(* Logix 5000 project; controller default_profile 5069-L306ERM rev 31.11; software revision 31.01 *)

TASK MainTask (continuous, watchdog 500 ms) : MainProgram

MODULES
   Local : 5069-L306ERM (5069 0, rev 31.11)
       : 5069-IB16 (5069 2, rev 2.14, StandardDataDriven RPI 5 ms)
       : vendor 1 type 7 code 1213 (5069 1, rev 3.14, StandardDataDriven RPI 5 ms)
END_MODULES

VAR_GLOBAL   (* controller tags *)
   Heater_Blower : BOOL;
   Load_Cell : DINT;
   Motor1_Backwards : BOOL;
   Motor1_Forwards : BOOL;
   Motor2 : BOOL;
   Motor_Timer : TIMER := (PRE := 2000);
   Piston : BOOL;
   Piston_Timer : TIMER := (PRE := 10);
   Platform_1 : DINT;
   Platform_2 : DINT := 1000000;
   Platform_3 : DINT := 2000000;
   Position : DINT;
   Radians : DINT;
   Rotation : DINT;
   RUN : BOOL;
   STANDBY : BOOL := 1;
   START : BOOL;
   STOP : BOOL;
   SV1 : BOOL;
   SV2 : BOOL;
   Task : DINT;
   Timer1 : TIMER := (PRE := 6000);
   Timer2 : TIMER := (PRE := 25000);
END_VAR

PROGRAM MainProgram   (* main routine MainRoutine *)

ROUTINE MainRoutine   (* ladder *)
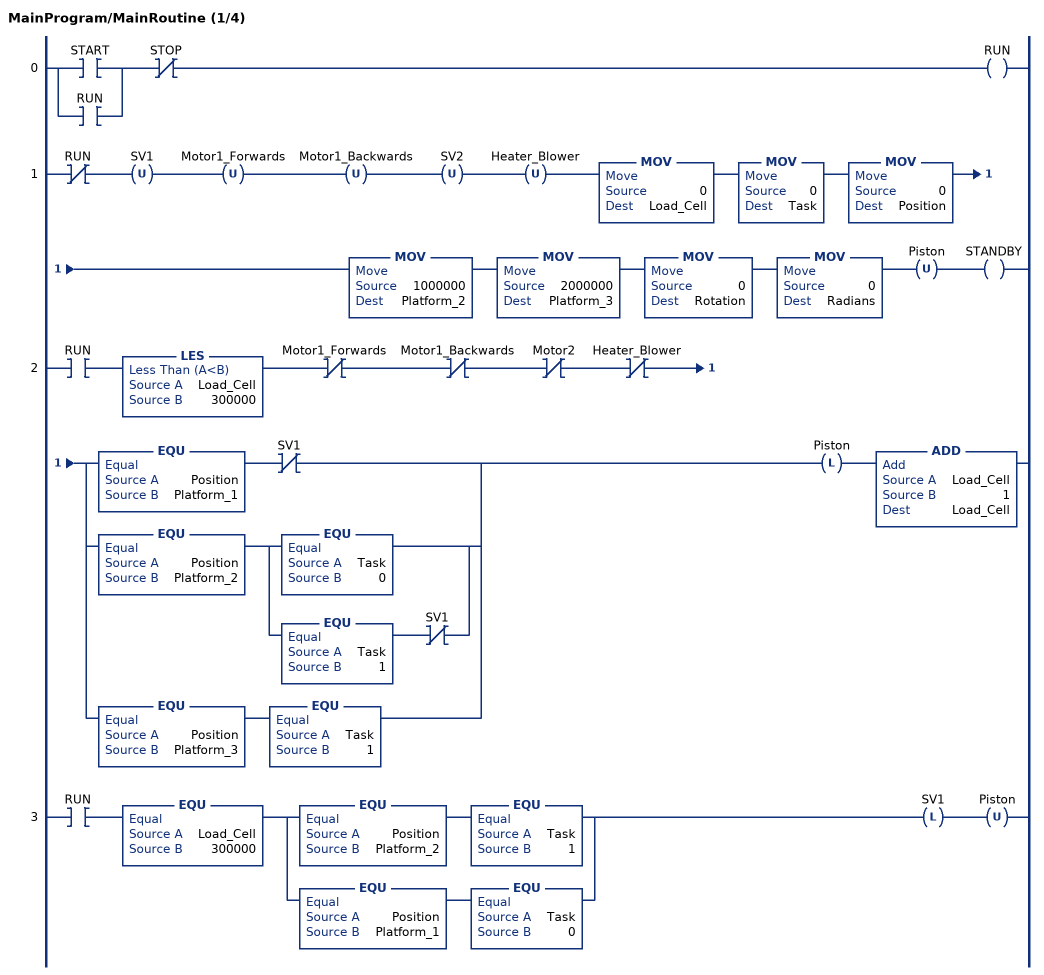
   0: [XIC(START) ,XIC(RUN) ]XIO(STOP)OTE(RUN);
   1: XIO(RUN)OTU(SV1)OTU(Motor1_Forwards)OTU(Motor1_Backwards)OTU(SV2)OTU(Heater_Blower)MOV(0,Load_Cell)MOV(0,Task)MOV(0,Position)MOV(1000000,Platform_2)MOV(2000000,Platform_3)MOV(0,Rotation)MOV(0,Radians)OTU(Piston)OTE(STANDBY);
   2: XIC(RUN)LES(Load_Cell,300000)XIO(Motor1_Forwards)XIO(Motor1_Backwards)XIO(Motor2)XIO(Heater_Blower)[EQU(Position,Platform_1) XIO(SV1) ,[EQU(Position,Platform_2) [EQU(Task,0) ,EQU(Task,1) XIO(SV1) ] ,EQU(Position,Platform_3) EQU(Task,1) ] ]OTL(Piston)ADD(Load_Cell,1,Load_Cell);
   3: XIC(RUN)EQU(Load_Cell,300000)[EQU(Position,Platform_2) EQU(Task,1) ,EQU(Position,Platform_1) EQU(Task,0) ]OTL(SV1)OTU(Piston);
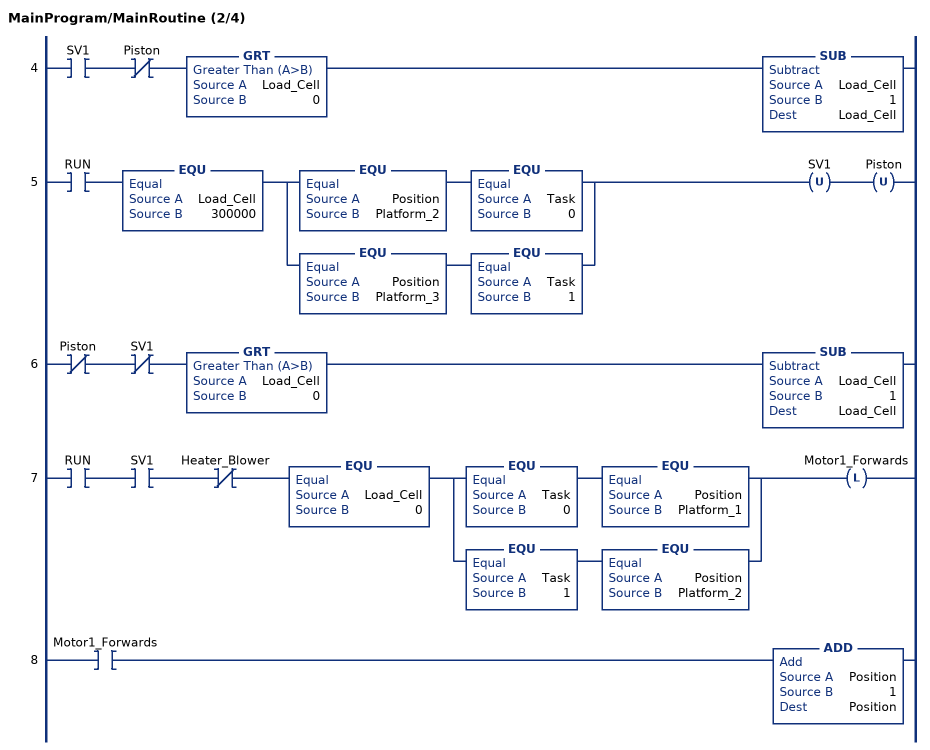
   4: XIC(SV1)XIO(Piston)GRT(Load_Cell,0)SUB(Load_Cell,1,Load_Cell);
   5: XIC(RUN)EQU(Load_Cell,300000)[EQU(Position,Platform_2) EQU(Task,0) ,EQU(Position,Platform_3) EQU(Task,1) ]OTU(SV1)OTU(Piston);
   6: XIO(Piston)XIO(SV1)GRT(Load_Cell,0)SUB(Load_Cell,1,Load_Cell);
   7: XIC(RUN)XIC(SV1)XIO(Heater_Blower)EQU(Load_Cell,0)[EQU(Task,0) EQU(Position,Platform_1) ,EQU(Task,1) EQU(Position,Platform_2) ]OTL(Motor1_Forwards);
   8: XIC(Motor1_Forwards)ADD(Position,1,Position);
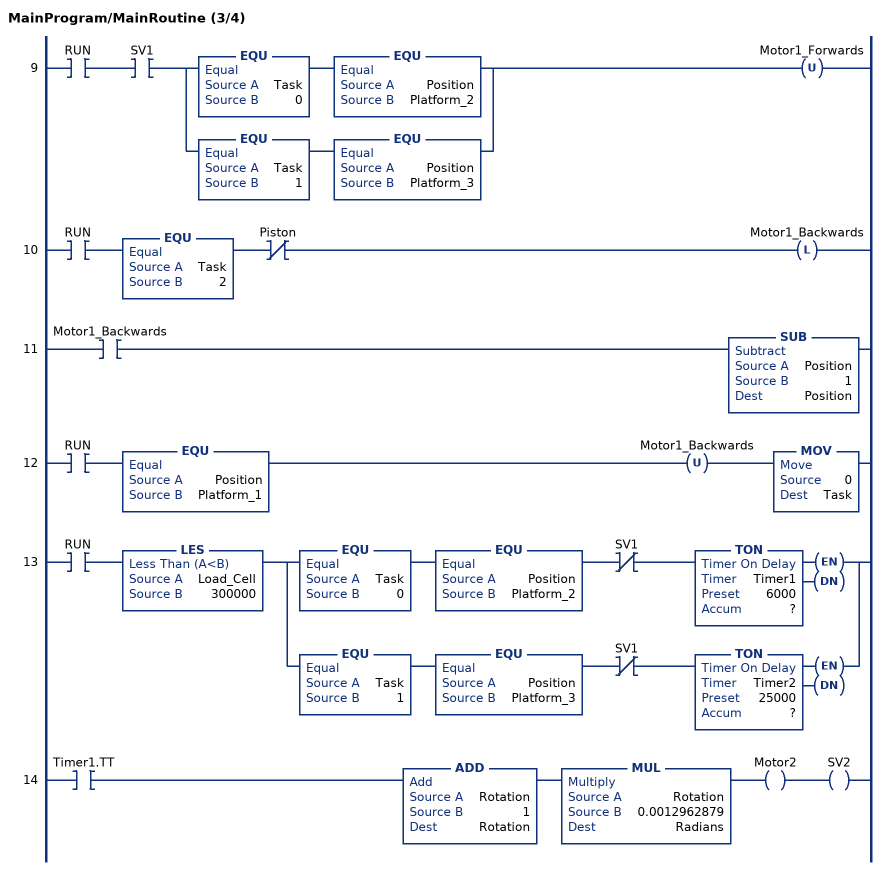
   9: XIC(RUN)XIC(SV1)[EQU(Task,0) EQU(Position,Platform_2) ,EQU(Task,1) EQU(Position,Platform_3) ]OTU(Motor1_Forwards);
   10: XIC(RUN)EQU(Task,2)XIO(Piston)OTL(Motor1_Backwards);
   11: XIC(Motor1_Backwards)SUB(Position,1,Position);
   12: XIC(RUN)EQU(Position,Platform_1)OTU(Motor1_Backwards)MOV(0,Task);
   13: XIC(RUN)LES(Load_Cell,300000)[EQU(Task,0) EQU(Position,Platform_2) XIO(SV1) TON(Timer1,?,?) ,EQU(Task,1) EQU(Position,Platform_3) XIO(SV1) TON(Timer2,?,?) ];
   14: XIC(Timer1.TT)ADD(Rotation,1,Rotation)MUL(Rotation,0.0012962879,Radians)OTE(Motor2)OTE(SV2);
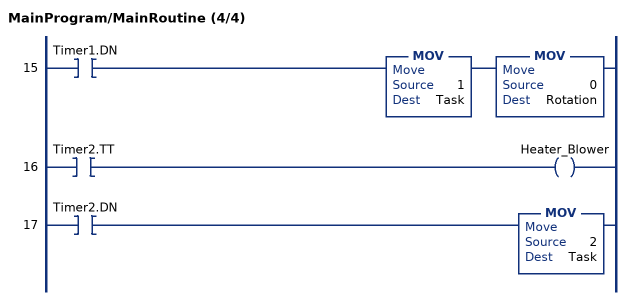
   15: XIC(Timer1.DN)MOV(1,Task)MOV(0,Rotation);
   16: XIC(Timer2.TT)OTE(Heater_Blower);
   17: XIC(Timer2.DN)MOV(2,Task);
END_ROUTINE
END_PROGRAM
